# EPICS substitutions: streamApp/pluginDb/pluginTransform.substitutions
#
# pluginTransform.substitutions
#

file NDTransform.template
{
	{
    PORT            = "Trans\$(N)",
    P               = "$(CAM):",
	R				= "$(PORT):",
    ADDR            = "\$(ADDR=0)",
    TIMEOUT         = "\$(TIMEOUT=1)",
    NDARRAY_PORT    = "\$(PLUGIN_SRC)",
    NDARRAY_ADDR    = "\$(NDARRAY_ADDR=0)",
	}
}
